Yaskawa INFORM job: BALON_1.JBI

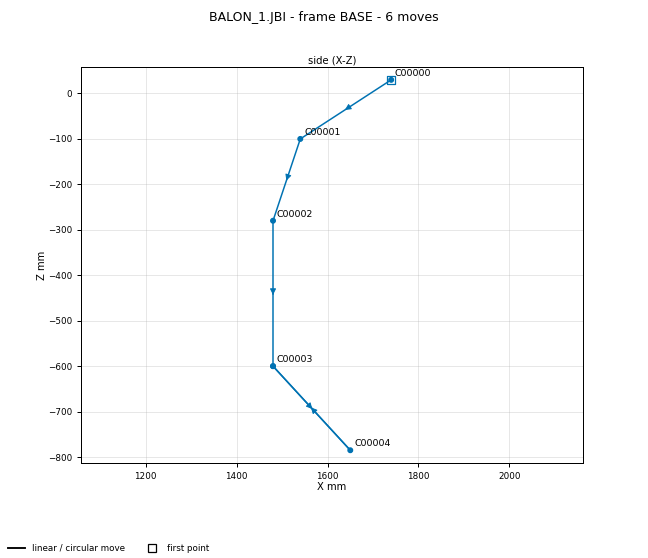
[picture p0: tool path of BALON_1.JBI in frame BASE, 6 of 6 moves have a stored position in this frame; points joined in program order, loops and branches not executed]
/JOB
//NAME BALON_1
//POS
///NPOS 6,0,6,0,0,0
///TOOL 0
///POSTYPE BASE
///RECTAN
///RCONF 0,0,0,0,0,0,0,0,0,0,0,0,0,0,0,0,0,0,0,0,0,0,0,0
C00000=1740.000,35.000,30.000,-180.0000,-30.0000,0.0000
C00001=1540.000,35.000,-100.000,180.0000,-50.0000,0.0000
C00002=1480.000,35.000,-280.000,-100.0000,-90.0000,-75.0000
C00003=1480.000,35.000,-600.000,-100.0000,-90.0000,-75.0000
C00004=1650.000,35.000,-785.000,-180.0000,-75.0000,0.0000
C00005=1480.000,35.000,-600.000,-100.0000,-90.0000,-75.0000
///POSTYPE PULSE
///PULSE
EC00000=0
EC00001=370000
EC00002=0
EC00003=370000
EC00004=0
EC00005=0
//INST
///DATE 2023/04/18 16:39
///ATTR SC,RW,RJ
////FRAME BASE
///GROUP1 RB1,ST1
NOP
MOVJ C00000 EC00000 VJ=15.00
CALL JOB:SPYON
MOVL C00001 EC00001 V=200.0
MOVL C00002 EC00002 V=200.0
MOVL C00003 EC00003 V=200.0
MOVL C00004 EC00004 V=200.0
CALL JOB:SPYOF
MOVL C00005 EC00005 V=200.0
END
